INTERFACE IHeartBeat EXTENDS __SYSTEM.IQueryInterface

PROPERTY GetErrorMessage : T_MaxString;
GET
END_GET
END_PROPERTY

//actual Heartbeat of PLC
PROPERTY GetHeartBeat : UINT
GET
END_GET
END_PROPERTY

PROPERTY GetHeartbeatTimeoutTime : TIME
GET
END_GET
END_PROPERTY

PROPERTY GetState : eHeartBeatState
GET
END_GET
END_PROPERTY

METHOD IncreaseHeartBeat : UINT
VAR_INPUT
    externalHeartBeat : UINT;
END_VAR
END_METHOD

END_INTERFACE

(* stored: Version 1.1.0.1, ProductVersion 3.1.4024.12
   Itf IHeartBeat: Id {91448687-689a-4ab3-9ef3-21f38db9796a}
   Property GetErrorMessage: Id {69c031b9-aefa-4d4b-a8cf-a96d5c13d03f}
   Get Get: Id {1ab98fdd-ac77-4486-8b8a-b0183f154cc1}
   Property GetHeartBeat: Id {f6c088ce-333c-4776-8a3c-5a7c4fa1691d}
   Get Get: Id {02911b99-b9ca-4180-9d7f-4cb2e7fd7847}
   Property GetHeartbeatTimeoutTime: Id {11df7e1c-b9a9-4a09-b6de-9de3fd4ebcf8}
   Get Get: Id {1c5c5f70-a0f8-4618-b225-591fb617cfc5}
   Property GetState: Id {f029fddf-911a-41cb-92f7-e1e515c28dd5}
   Get Get: Id {1fc311b5-5681-4098-b262-8f36d6a388a6}
   Method IncreaseHeartBeat: Id {ac456990-abbb-42a9-9cb3-a4c41faab5f9} *)
